FUNCTION SuctionQualityPtr  : BOOL
VAR_INPUT
	suctions : POINTER TO SuctionPad;
	numPads : DINT;
END_VAR
VAR_INPUT
	insertionMaterial : STRING;
	recipeMaterial : STRING;
END_VAR
VAR
	i : DINT;
	
	failedVacuums : INT;
	numVacuums : INT;
END_VAR

(*
IF insertionMaterial <> recipeMaterial THEN //reintroduce this condition later
	RETURN;
END_IF
*)

FOR i:=0 TO numPads BY 1 DO
	IF suctions[i].enable THEN
		numVacuums := numVacuums + 1;
		IF NOT suctions[i].occupied THEN
			failedVacuums := failedVacuums + 1;
		END_IF
	END_IF
	
END_FOR

//SuctionQualityPtrArr := failedVacuums < (numVacuums * 1/3);
SuctionQualityPtr := TRUE;

END_FUNCTION

(* stored: Version 1.1.0.1, ProductVersion 3.1.4024.11
   POU SuctionQualityPtr: Id {ac8e9afb-0ca2-4faa-aa99-c7323dd4df65}, SpecialFunc None *)
